# EPICS IOC start-up script: iocBoot/common/init_bkh_odm.iocsh
# Beckhoff config for ODM sensor cell type (oldham)
# 20210401 mdunning
#
# Required macros:
#  BKH_PORT - Asyn port name
#  BKH_IP - Bus coupler node name or IP address
#
# This file should be executed from the ioc shell like so:
#  iocshLoad(filename, macros)
#  For example:
#  iocshLoad("$(TOP)/iocBoot/common/init_bkh_ms02.iocsh", "BKH_PORT=BKH02,BKH_IP=apc-sys0-ms02")

drvAsynIPPortConfigure("$(BKH_PORT)", "$(BKH_IP):502", 0,0,1)
modbusInterposeConfig("$(BKH_PORT)", 0, 1000)
drvMBusConfig("$(BKH_PORT)", 0, 0, 125, 0, "$(BKH_PORT)", 10)
#
# drvBkhAsynConfig(mbus_name, id, port, func, addr, len, nch, msec)
# mbus_name is a unique idendifier for bus couplers
# id is a unique module type identifier: 0 - coupler, 1 - analogSigned,
#     2 - analogUnsigned, 3 - digitalIn, 4 - digitalOut, 5 - motor.
# port is the asyn port name for the driver (pick a unique short name for each module as below)
# func is the modbus function (e.g. 5 - digitalOut, 2 - digitalIn, 3 - analog In/Out)
# addr is the modbus starting address of the memory image (group all modules of the same modbus function together)
# len is the length of the memory image, in bits (digital modules) or 16 bit words (analog modules)
# nch is the number of channels
# msec is poll routine timeout in milliseconds
#
# These are standard bus coupler commands
drvBkhAsynConfig("$(BKH_PORT)", 0,   "$(BKH_PORT)_DEBUG", 3,      0, 125,  2,    0)
drvBkhAsynConfig("$(BKH_PORT)", 0,   "$(BKH_PORT)_B900R", 3, 0x1000,  33, 33,    0)
drvBkhAsynConfig("$(BKH_PORT)", 0,   "$(BKH_PORT)_B900W", 3, 0x110a,  26, 26,    0)
#
# These are for the bus terminals
drvBkhAsynConfig("$(BKH_PORT)", 2, "$(BKH_PORT)_3012_01", 3,      0,   4,  2,  250)

#asynSetTraceIOMask("$(BKH_PORT)_3012_01", 0, 4)
#asynSetTraceMask("$(BKH_PORT)_3012_01", 0, 0x9)

# End of file
